FUNCTION_BLOCK tripTest (* Basic Function Block Type *)
  (* Standard: 61499-2 *)
  (* Version 0.0, 7/4/2016, gulzha, nxtControl GmbH, Template *)
  PACKAGE Main;
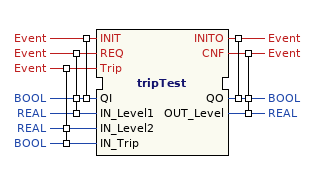
  EVENT_INPUT
    INIT WITH QI; (* Initialization Request *)
    REQ WITH QI, IN_Level1; (* Normal Execution Request *)
    Trip WITH IN_Level2, IN_Trip;
  END_EVENT
  EVENT_OUTPUT
    INITO WITH QO; (* Initialization Confirm *)
    CNF WITH QO, OUT_Level; (* Execution Confirmation *)
  END_EVENT
  VAR_INPUT
    QI : BOOL; (* Input event qualifier *)
    IN_Level1 : REAL;
    IN_Level2 : REAL;
    IN_Trip : BOOL;
  END_VAR
  VAR_OUTPUT
    QO : BOOL; (* Output event qualifier *)
    OUT_Level : REAL;
  END_VAR
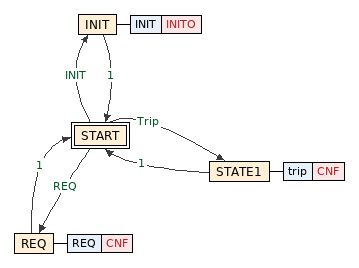
  EC_STATES
    START; (* Initial State *)
    INIT : INIT -> INITO; (* Initialization *)
    REQ : REQ -> CNF; (* Normal execution *)
    STATE1 : trip -> CNF;
  END_STATES
  EC_TRANSITIONS
    START TO INIT := INIT;
    INIT TO START := 1;
    START TO REQ := REQ;
    REQ TO START := 1;
    START TO STATE1 := Trip;
    STATE1 TO START := 1;
  END_TRANSITIONS
  ALGORITHM INIT IN ST: (* Initialization algorithm *)
;
  END_ALGORITHM
  ALGORITHM REQ IN ST: (* Normally executed algorithm *)
;

OUT_Level:=IN_Level1;
  END_ALGORITHM
  ALGORITHM trip IN ST:
;
IF (IN_Trip) THEN
	OUT_Level:=IN_Level2;
END_IF;
  END_ALGORITHM
END_FUNCTION_BLOCK
